// TwinCAT 3 PLC project TCP_IP
// ProgramVersion: 3.1.4023.0
// libraries:
//   Tc2_Standard, * (Beckhoff Automation GmbH)
//   Tc2_System, * (Beckhoff Automation GmbH)
//   Tc2_TcpIp, * (Beckhoff Automation GmbH)
//   Tc2_Utilities, * (Beckhoff Automation GmbH)
//   Tc3_JsonXml, * (Beckhoff Automation GmbH)
//   Tc3_Module, * (Beckhoff Automation GmbH)
// project tree:
//   DUTs/ sensorData.TcDUT
//   / GlobalTextList.TcGTLO, PlcTask.TcTTO, Visualization Manager.TcVMO (not stored)
//   POUs/ JSON_decode.TcPOU, MAIN.TcPOU, tcp_ip.TcPOU
//   VISUs/ Visualization.TcVIS
// real-time tasks:
//   TASK PlcTask: cycle T#10ms, priority 20, ADS port 350

CONFIGURATION TCP_IP
    RESOURCE PLC ON TwinCAT3
        TASK PlcTask(INTERVAL := T#10ms, PRIORITY := 20);
        PROGRAM MAIN WITH PlcTask : MAIN;
    END_RESOURCE
END_CONFIGURATION

// ---- DUTs/sensorData.TcDUT
TYPE sensorData :
STRUCT
	id			: STRING(20);
	flag		: DINT; 
	mode		: DINT;
	temp		: DINT;
	hum			: DINT;
	battery		: DINT;
END_STRUCT
END_TYPE

// ---- POUs/MAIN.TcPOU
PROGRAM MAIN
VAR
END_VAR

JSON_decode();

END_PROGRAM

// ---- POUs/JSON_decode.TcPOU
PROGRAM JSON_decode
VAR
	mydata : sensorData;
	fixedMessage : STRING(150) := '{"id": "4CCE8E","battery": 80,"flag": 0,"mode": 1,"temp": 23,"hum": 0}';
	//block
	fbJson		: FB_JsonDomParser;
	//parsed
	parsedDoc	: SJsonValue;
	parsedVal	: SJsonValue;

END_VAR

// rx
parsedDoc := fbJson.ParseDocument(fixedMessage);

parsedVal := fbJson.FindMember(parsedDoc, 'id');
mydata.id := fbJson.GetString(parsedVal);

parsedVal := fbJson.FindMember(parsedDoc, 'battery');
mydata.battery := fbJson.GetInt(parsedVal);

parsedVal := fbJson.FindMember(parsedDoc, 'flag');
mydata.flag := fbJson.GetInt(parsedVal);

parsedVal := fbJson.FindMember(parsedDoc, 'mode');
mydata.mode := fbJson.GetInt(parsedVal);

parsedVal := fbJson.FindMember(parsedDoc, 'temp');
mydata.temp := fbJson.GetInt(parsedVal);

parsedVal := fbJson.FindMember(parsedDoc, 'hum');
mydata.hum := fbJson.GetInt(parsedVal);
(*
parsedVal2 := fbJson.FindMember(parsedVal1, 'battery');
mydata.battery := fbJson.GetString(parsedVal);

parsedVal3 := fbJson.FindMember(parsedVal2, 'flag');
mydata.flag := fbJson.GetString(parsedVal);

parsedVal4 := fbJson.FindMember(parsedVal3, 'mode');
mydata.mode := fbJson.GetString(parsedVal);

parsedVal5 := fbJson.FindMember(parsedVal4, 'temp');
mydata.temp := fbJson.GetString(parsedVal);

parsedVal6 := fbJson.FindMember(parsedVal5, 'hum');
mydata.hum := fbJson.GetString(parsedVal);*)

END_PROGRAM

// ---- POUs/tcp_ip.TcPOU
PROGRAM tcp_ip
VAR
	bConnect : BOOL;
	bRecieve : BOOL;
	FB_create : FB_SocketUdpCreate;
	FB_Recieve: FB_SocketUdpReceiveFrom;
	FB_close  : FB_SocketClose;
	FB_info	  : FB_GetAdaptersInfo;
	data: ARRAY[0..5000] OF BYTE;
END_VAR

FB_info(
sNetID := ,
tTimeout := T#5S);

FB_create(
	sSrvNetId:= , 							//Lokaal netwerk (mag leeg blijven)
	sLocalHost:= '192.168.1.157', 			//Eigen ip van de PC en ingesteld in de gateway
	nLocalPort:= 25565,						//Ingesteld op de gateway
	bExecute:= bConnect,					//Trigger voor functieblok
	tTimeout:= T#10S);


FB_Recieve(
	sSrvNetId:= , 									//Lokaal netwerk (mag leeg blijven)
	hSocket:= FB_create.hSocket,					 
	cbLen:= SIZEOF(data), 							//Kijkt naar de lengte van het bericht
	pDest:= ADR(data), 								//Plaat waar de het bericht wordt opgeslaan
	bExecute:= NOT FB_recieve.bBusy AND bRecieve, 	//Trigger voor functieblok
	tTimeout:= T#10S);
	
FB_close(
	sSrvNetId:= , 							//Lokaal netwerk (mag leeg blijven)
	hSocket:= FB_create.hSocket, 			
	bExecute:= NOT bConnect, 				//Sluiten van de connectie 
	tTimeout:= T#1S);

END_PROGRAM

// ---- GlobalTextList.TcGTLO
TEXTLIST GlobalTextList
  383 = '%'
  151 = '%id'
  174 = '%s'
  135 = 'battery: %s'
  425 = 'flag: %s'
  597 = 'humidity: %s'
  585 = 'id %s'
  295 = 'id: %s'
  676 = 'JSON_decode:id'
  422 = 'mode: %s'
  245 = 'temperature: %s'
END_TEXTLIST

// ---- VISUs/Visualization.TcVIS
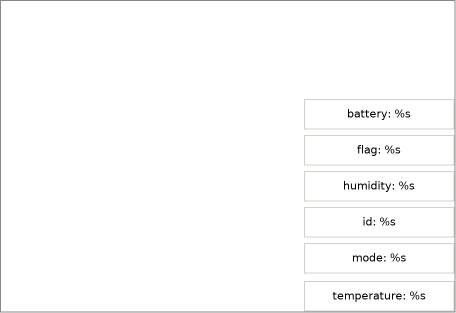
VISUALIZATION Visualization  // 456x313
    Textfield (304,99 150x30), "battery: %s", text variable: JSON_decode.mydata.battery
    Textfield (304,135 150x30), "flag: %s", text variable: JSON_decode.mydata.flag
    Textfield (304,171 150x30), "humidity: %s", text variable: JSON_decode.mydata.hum
    Textfield (304,207 150x30), "id: %s", text variable: JSON_decode.mydata.id
    Textfield (304,243 150x30), "mode: %s", text variable: JSON_decode.mydata.mode
    Textfield (304,281 150x30), "temperature: %s", text variable: JSON_decode.mydata.temp
END_VISUALIZATION
